{attribute 'GeneratedUsingTerminal: EP6002-0002-0017'}
{attribute addProperty BoxType "EP6002-0002-0017"}
{attribute addProperty Id "StatusAT %I*WORD2Data_InAT %I*ARRAY[0..21] OF USINT22"}
{attribute addProperty CRC "3532970676"}
{attribute addProperty Size "24"}
TYPE COM_TxPDO_Map_Inputs_Channel_C252EAC2 :
STRUCT
	{attribute addProperty Name "Status"}
	Status AT %I* : WORD;
	{attribute addProperty Name "Data_In"}
	Data_In AT %I* : ARRAY[0..21] OF USINT;
END_STRUCT
END_TYPE

(* stored: Version 1.2.0.0, ProductVersion 3.1.4024.9
   DUT COM_TxPDO_Map_Inputs_Channel_C252EAC2: Id {f8f64458-8527-4c34-ac4e-e3579e85f704} *)
